// TIA Portal project "Milling Cutter With Extraction" (V15)

(* hardware
DEVICE "S7-1200 station_1"  S7-1200 Station
   slot 0: "Rack_0"  S7-1200 Rack  Rack  V1.0
   slot 1: "PLC_1"  CPU 1214C AC/DC/Rly  6ES7 214-1BG40-0XB0  V4.2
*)

// ===== PLC "PLC_1"  CPU 1214C AC/DC/Rly =====

VAR_GLOBAL   // PLC tag table "Tag table_1"
   "ESO" AT %I0.0 : Bool;   // NC
   "S ON (M)" AT %I0.1 : Bool;   // Mill Switch NO
   "S OFF" AT %I0.3 : Bool;   // NC
   "F (M)" AT %I0.4 : Bool;   // Mill Relay NC
   "F (E)" AT %I0.5 : Bool;   // Ext Relay NC
   "Q (M)" AT %Q0.0 : Bool;   // Milling Motor Contactor
   "Q (E)" AT %Q0.1 : Bool;   // Extraction Motor Contactor
   "P (M)" AT %Q0.2 : Bool;   // Milling Working Lamp
   "P (E)" AT %Q0.3 : Bool;   // Extraction Working Lamp
   "P (F)" AT %Q0.4 : Bool;   // Fault Lamp
   "S ON (E)" AT %I0.2 : Bool;   // Ext Switch NO
   "S Reset" AT %I0.6 : Bool;   // Reset ESO
   "F Reset" AT %Q0.5 : Bool;   // Hold reset
END_VAR

ORGANIZATION_BLOCK "Main"   // OB1, LAD, ProgramCycle
TITLE = "Main Program Sweep (Cycle)"
{ S7_Optimized_Access := 'TRUE' }
VERSION : 0.1
   VAR_INPUT
      Initial_Call : Bool;   // Initial call of this OB
      Remanence : Bool;   // =True, if remanent data are available
   END_VAR
BEGIN

REGION Network 1: Extraction Motor Contactor
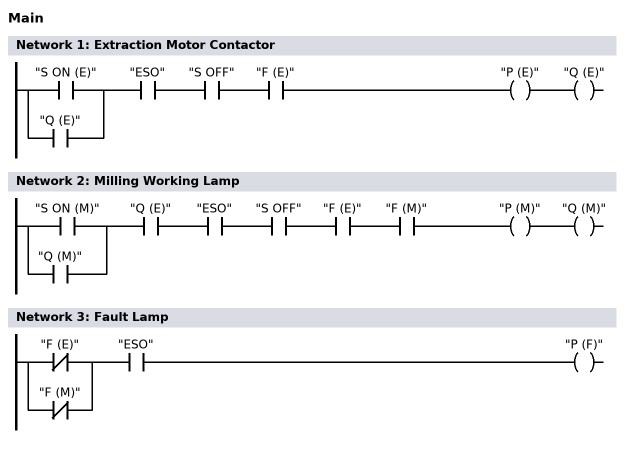
   RUNG wire#powerrail
      Contact( "S ON (E)" )
      wire#w1
      Contact( "ESO" )
      Contact( "S OFF" )
      Contact( "F (E)" )
      Coil( "P (E)" )
      Coil( "Q (E)" )
   END_RUNG
   RUNG wire#powerrail
      Contact( "Q (E)" )
   END_RUNG wire#w1
   // the same network as SCL:
   "P (E)" := ("S ON (E)" OR "Q (E)") AND "ESO" AND "S OFF" AND "F (E)";
   "Q (E)" := "P (E)";
END_REGION

REGION Network 2: Milling Working Lamp
   RUNG wire#powerrail
      Contact( "S ON (M)" )
      wire#w1
      Contact( "Q (E)" )
      Contact( "ESO" )
      Contact( "S OFF" )
      Contact( "F (E)" )
      Contact( "F (M)" )
      Coil( "P (M)" )
      Coil( "Q (M)" )
   END_RUNG
   RUNG wire#powerrail
      Contact( "Q (M)" )
   END_RUNG wire#w1
   // the same network as SCL:
   "P (M)" := ("S ON (M)" OR "Q (M)") AND "Q (E)" AND "ESO" AND "S OFF" AND "F (E)" AND "F (M)";
   "Q (M)" := "P (M)";
END_REGION

REGION Network 3: Fault Lamp
   RUNG wire#powerrail
      I_Contact( "F (E)" )
      wire#w1
      Contact( "ESO" )
      Coil( "P (F)" )
   END_RUNG
   RUNG wire#powerrail
      I_Contact( "F (M)" )
   END_RUNG wire#w1
   // the same network as SCL:
   "P (F)" := (NOT "F (E)" OR NOT "F (M)") AND "ESO";
END_REGION
END_ORGANIZATION_BLOCK